// TIA Portal V20 export
DATA_BLOCK "DB_AnalogInputAction"   // DB1304
TITLE = TEMPERATURE SETTINGS
{ S7_Optimized_Access := 'FALSE'; DB_Accessible_From_OPC_UA := 'FALSE' }
AUTHOR : SAN
// stored: AutoNumber false, DBAccessibleFromOPCUA false, DBAccessibleFromWebserver false
   VAR
      Laser_Power_Meter : "AnalogInAction_DT";
      Axis_B_Clamping_Part : "AnalogInAction_DT";
      Laser_Air_Pressure_Process : "AnalogInAction_DT";
      Inlet_Air_Pressure : "AnalogInAction_DT";
      Ambiant_Temperature : "AnalogInAction_DT";
      Machine_Temperature : "AnalogInAction_DT";
      Cold_Water_Temperature_Input : "AnalogInAction_DT";
      Cold_Water_Temperature_Output : "AnalogInAction_DT";
      X_Axis_Temperature_PT1000 : "AnalogInAction_DT";
      Y_Axis_Temperature_PT1000 : "AnalogInAction_DT";
      X_Axis_Temperature_PTC : "AnalogInAction_DT";
      Y_Axis_Temperature_PTC : "AnalogInAction_DT";
      Nozzle_Overpressure : "AnalogInAction_DT";
      Optical_Path_Overpressure : "AnalogInAction_DT";
      Laser_Head_Overpressure : "AnalogInAction_DT";
      ZL_Axis_Overpressure : "AnalogInAction_DT";
      XY_Axis_Overpressure : "AnalogInAction_DT";
      Left_Aspiration : "AnalogInAction_DT";
      Right_Aspiration : "AnalogInAction_DT";
      Free_IW458 : "AnalogInAction_DT";
      Clim_Temperature : "AnalogInAction_DT";
      Free_IW482 : "AnalogInAction_DT";
      Free_IW484 : "AnalogInAction_DT";
      Free_IW486 : "AnalogInAction_DT";
      Sensor_Controller_Station1 : "AnalogInAction_DT";
      Cabinet_Temperature : "AnalogInAction_DT";
      Free_IW464 : "AnalogInAction_DT";
      Free_IW466 : "AnalogInAction_DT";
   END_VAR
BEGIN
   Laser_Power_Meter.ID_Measure := 1;
   Axis_B_Clamping_Part.ID_Measure := 2;
   Laser_Air_Pressure_Process.ID_Measure := 3;
   Inlet_Air_Pressure.ID_Measure := 4;
   Ambiant_Temperature.ID_Measure := 5;
   Machine_Temperature.ID_Measure := 6;
   Cold_Water_Temperature_Input.ID_Measure := 7;
   Cold_Water_Temperature_Output.ID_Measure := 8;
   X_Axis_Temperature_PT1000.ID_Measure := 9;
   Y_Axis_Temperature_PT1000.ID_Measure := 10;
   X_Axis_Temperature_PTC.ID_Measure := 11;
   Y_Axis_Temperature_PTC.ID_Measure := 12;
   Nozzle_Overpressure.ID_Measure := 13;
   Optical_Path_Overpressure.ID_Measure := 14;
   Laser_Head_Overpressure.ID_Measure := 15;
   ZL_Axis_Overpressure.ID_Measure := 16;
   XY_Axis_Overpressure.ID_Measure := 17;
   Left_Aspiration.ID_Measure := 18;
   Right_Aspiration.ID_Measure := 19;
   Free_IW458.ID_Measure := 20;
   Clim_Temperature.ID_Measure := 21;
   Free_IW482.ID_Measure := 22;
   Free_IW484.ID_Measure := 23;
   Free_IW486.ID_Measure := 24;
   Sensor_Controller_Station1.ID_Measure := 25;
   Cabinet_Temperature.ID_Measure := 26;
   Free_IW464.ID_Measure := 27;
   Free_IW466.ID_Measure := 28;
END_DATA_BLOCK
